{attribute 'linkalways'} 
{attribute 'no_explicit_call' := 'This FB is a CLASS and must be accessed using methods or properties'}
{attribute 'enable_dynamic_creation'}
FUNCTION_BLOCK Dictionary
VAR
	root : I_DictionaryTreeNode;
END_VAR

METHOD PUBLIC AddOrUpdate
VAR_INPUT
	Key : T_MAXSTRING;
	Value : ANY;
END_VAR
root := this^.RecursiveInsert(Key, Value, root);
END_METHOD

METHOD PRIVATE Balance : I_DictionaryTreeNode
VAR_INPUT
	Node : I_DictionaryTreeNode;
END_VAR
VAR
	balanceFactor : DINT;
END_VAR
balanceFactor := THIS^.GetBalanceFactor(Node);

IF (balanceFactor > 1) THEN
  IF (THIS^.getBalanceFactor(Node.left) < 0) THEN
	Node.left := THIS^.leftRotate(Node.left);
  END_IF
  Balance := THIS^.rightRotate(Node);
  RETURN;
END_IF

IF (balanceFactor < -1) THEN
  IF (THIS^.getBalanceFactor(Node.right) > 0) THEN
	Node.right := THIS^.rightRotate(Node.right);
  END_IF
  Balance := THIS^.leftRotate(Node);
  RETURN;
END_IF

Balance := Node;
END_METHOD

METHOD PUBLIC Clear
VAR_INPUT
END_VAR
THIS^.RecursiveClear(root);
root := 0;
END_METHOD

METHOD PUBLIC ContainsKey : BOOL
VAR_INPUT
	Key : T_MAXSTRING;
END_VAR
VAR
	foundNode : I_DictionaryTreeNode;
END_VAR
foundNode := THIS^.RecursiveFind(Key, root);

IF foundNode = 0 THEN
	RETURN;
END_IF

ContainsKey := TRUE;
END_METHOD

METHOD PRIVATE FindMinimum : I_DictionaryTreeNode
VAR_INPUT
	Node : I_DictionaryTreeNode;
END_VAR
VAR
	nextNode : I_DictionaryTreeNode;
END_VAR
nextNode := Node;

WHILE (nextNode.left <> 0) DO
      nextNode := nextNode.left;
END_WHILE;

FindMinimum := nextNode;
END_METHOD

METHOD PRIVATE GetBalanceFactor : DINT
VAR_INPUT
	Node : I_DictionaryTreeNode;
END_VAR
GetBalanceFactor := THIS^.GetHeight(node.left) - THIS^.GetHeight(node.right);
END_METHOD

METHOD PRIVATE GetHeight : DINT
VAR_INPUT
	Node : I_DictionaryTreeNode;
END_VAR
IF Node = 0 THEN
	GetHeight := 0;
	RETURN;
END_IF

GetHeight := Node.Height;
END_METHOD

METHOD PRIVATE LeftRotate : I_DictionaryTreeNode
VAR_INPUT
	Node : I_DictionaryTreeNode;
END_VAR
VAR
	newRoot : I_DictionaryTreeNode;
END_VAR
newRoot := Node.right;
Node.right := newRoot.left;
newRoot.left := Node;
THIS^.UpdateHeight(Node);
THIS^.UpdateHeight(newRoot);
LeftRotate := newRoot;
END_METHOD

METHOD PRIVATE RecursiveClear
VAR_INPUT
	Node : I_DictionaryTreeNode;
END_VAR
IF (Node = 0) THEN
	RETURN;
END_IF

RecursiveClear(Node.Left);
RecursiveClear(Node.Right);
Node.Dispose();
END_METHOD

METHOD PRIVATE RecursiveDelete : I_DictionaryTreeNode
VAR_INPUT
	Key : T_MAXSTRING;
	Node : I_DictionaryTreeNode;
	Parent : I_DictionaryTreeNode;
END_VAR
VAR
	newNode : I_DictionaryTreeNode; 
	parentNode : I_DictionaryTreeNode;
	minValueNode : I_DictionaryTreeNode;
	minValueNodeParent : I_DictionaryTreeNode;
END_VAR
parentNode := Parent;

IF (Node = 0) THEN
	RETURN;
END_IF

IF (Key < Node.Key) THEN
	parentNode := Node;
	Node.left := THIS^.RecursiveDelete(Key, Node.left, parentNode);
ELSIF (Key > Node.Key) THEN
	parentNode := node;
	Node.right := THIS^.RecursiveDelete(Key, Node.right, parentNode);
ELSE 
	// Case 1: Node with only one child or no child
	IF (Node.Left = 0) OR (Node.Right = 0) THEN
		
		IF (Node.Left = 0) THEN
			newNode := Node.Right;
		ELSE
			newNode := Node.Left;
		END_IF
	
		IF (parentNode <> 0) THEN
			IF (parentNode.left = Node) THEN
				parentNode.left := newNode;
			ELSE 
				parentNode.right := newNode;
			END_IF
		END_IF
		
		Node.Dispose();
		RecursiveDelete.Delete := newNode;
		RETURN;
		
	END_IF

	// Case 2: Node with two children
	minValueNode := THIS^.FindMinimum(Node.Right);
	minValueNodeParent := THIS^.RecursiveFindParent(minValueNode.Key, THIS^.root, 0);
	
	IF (minValueNode.Right <> 0) THEN
		minValueNodeParent.Left := minValueNode.Right;
	ELSE 
		minValueNodeParent.Left := 0;
	END_IF
	
	minValueNode.Left := Node.Left;
	minValueNode.Right := Node.Right;
	
	IF (parentNode <> 0) THEN
		IF (parentNode.left = Node) THEN
			parentNode.left := minValueNode;
		ELSE 
			parentNode.right := minValueNode;
		END_IF
	END_IF
	
	Node.Dispose();
	RecursiveDelete.Delete := minValueNode;
	RETURN;
END_IF

THIS^.updateHeight(Node);
RecursiveDelete.Delete := THIS^.balance(Node);
END_METHOD

METHOD PRIVATE RecursiveFind : I_DictionaryTreeNode
VAR_INPUT
	Key : T_MAXSTRING;
	Node : I_DictionaryTreeNode;
END_VAR
IF (Node = 0) THEN
	RETURN;
END_IF

IF (Key < Node.key) THEN
  RecursiveFind := THIS^.RecursiveFind(key, Node.left);
  RETURN;
ELSIF (key > Node.key) THEN
  RecursiveFind := THIS^.RecursiveFind(key, Node.right);
  RETURN;
ELSE 
  RecursiveFind := Node;
  RETURN;
END_IF
END_METHOD

METHOD PRIVATE RecursiveFindParent : I_DictionaryTreeNode
VAR_INPUT
	Key : T_MAXSTRING;
	Node : I_DictionaryTreeNode;
	Parent : I_DictionaryTreeNode;
END_VAR
IF (Node = 0) THEN
	RETURN;
END_IF

IF (Key < Node.Key) THEN
	RecursiveFindParent := THIS^.RecursiveFindParent(Key, Node.Left, Node);
	RETURN;
ELSIF (Key > Node.Key) THEN
	RecursiveFindParent :=  THIS^.RecursiveFindParent(Key, Node.Right, Node);
	RETURN;
ELSE 
	RecursiveFindParent := Parent;
END_IF
END_METHOD

METHOD PRIVATE RecursiveInsert : I_DictionaryTreeNode
VAR_INPUT
	Key : T_MAXSTRING;
	Value : ANY;
	Node : I_DictionaryTreeNode;
END_VAR
VAR
	pAVLTreeNode : POINTER TO DictionaryTreeNode;
END_VAR
IF (Node = 0) THEN
	pAVLTreeNode := __NEW(DictionaryTreeNode);
	pAVLTreeNode^.Initialize(Key, Value);
	RecursiveInsert := pAVLTreeNode^;
	RETURN;
END_IF

IF (Key < node.key) THEN
	Node.left := THIS^.RecursiveInsert(Key, Value, Node.left);
ELSIF (key > node.key) THEN
	Node.right := THIS^.RecursiveInsert(Key, Value, Node.right);
ELSE
	Node.Initialize(Key,Value);
END_IF

THIS^.updateHeight(node);
RecursiveInsert := THIS^.balance(node);
END_METHOD

METHOD PUBLIC Remove
VAR_INPUT
	Key : T_MAXSTRING;
END_VAR
root := THIS^.RecursiveDelete(Key, root, 0);
END_METHOD

METHOD PRIVATE RightRotate : I_DictionaryTreeNode
VAR_INPUT
	Node : I_DictionaryTreeNode;
END_VAR
VAR
	newRoot : I_DictionaryTreeNode;
END_VAR
newRoot := Node.left;
Node.left := newRoot.right;
newRoot.right := Node;
THIS^.UpdateHeight(Node);
THIS^.UpdateHeight(newRoot);
RightRotate := newRoot;
END_METHOD

METHOD PUBLIC TryAdd : BOOL
VAR_INPUT
	Key : T_MAXSTRING;
	Value : ANY;
END_VAR
IF ContainsKey(Key) THEN
	RETURN;
END_IF
	  
THIS^.AddOrUpdate(Key, Value);
TryAdd := TRUE;
END_METHOD

METHOD PUBLIC TryGetValue : BOOL
VAR_INPUT
	Key : T_MAXSTRING;
	Destination	: ANY;
END_VAR
TryGetValue := TryGetValueTo(Key, Destination.pValue, DINT_TO_UDINT(Destination.diSize));
END_METHOD

METHOD PUBLIC TryGetValueTo : BOOL
VAR_INPUT
	Key : T_MAXSTRING;
	DestinationAddress : PVOID;
	DestinationSize : UDINT;
END_VAR
VAR
	foundNode : I_DictionaryTreeNode;
END_VAR
foundNode := THIS^.RecursiveFind(Key, root);

IF foundNode = 0 THEN
	RETURN;
END_IF

TryGetValueTo := foundNode.TryGetTo(DestinationAddress, DestinationSize);
END_METHOD

METHOD PRIVATE UpdateHeight
VAR_INPUT
	Node : I_DictionaryTreeNode;
END_VAR
Node.height := 1 + MAX(THIS^.GetHeight(Node.left), THIS^.GetHeight(Node.right));
END_METHOD

END_FUNCTION_BLOCK

(* stored: Version 1.1.0.1, ProductVersion 3.1.4024.12
   POU Dictionary: Id {031dc881-40c6-4324-9d62-c901951acf8a}, SpecialFunc None
   Folder Private: Id {9d25b7c8-1df3-4ed3-9572-63622da8d884}
   Method AddOrUpdate: Id {570f59cb-7938-4dac-8308-7b97aad37be6}
   Method Balance: Id {de35709f-49a6-4b93-a3ed-80e501fcabee}
   Method Clear: Id {9a75fda3-7d3e-4c00-8099-3ed82d8caa06}
   Method ContainsKey: Id {71cf2ebb-029b-4b77-a924-aa3f84d32e9a}
   Method FindMinimum: Id {4570296d-5467-479c-98b1-7fba065dc91f}
   Method GetBalanceFactor: Id {2a9ce396-eba7-4b31-8293-f5940b4357aa}
   Method GetHeight: Id {7b7a5b98-4d55-42ed-abb9-612f56324af2}
   Method LeftRotate: Id {1e3efb6c-46c1-4085-b7eb-b2d236432957}
   Method RecursiveClear: Id {e76039d0-529f-47ec-a7ab-8c3cbf1105bd}
   Method RecursiveDelete: Id {13a2f8bb-c070-4bfe-a28f-2d1a6438e9b8}
   Method RecursiveFind: Id {72c9c465-18ec-43f4-9bcd-fa5b73279ee3}
   Method RecursiveFindParent: Id {eb8edd98-ca1a-4ae6-8a6d-62c4cf4d7502}
   Method RecursiveInsert: Id {c57d1b55-65c3-4ee8-bbd0-7cf2e85e4be2}
   Method Remove: Id {f7e0145f-426d-4eb3-b5e3-9e9db70ed20a}
   Method RightRotate: Id {8508047b-6b5a-45a7-bfef-30c0ff9ccfee}
   Method TryAdd: Id {0579aed8-c227-47aa-b1a3-1246c4c9910b}
   Method TryGetValue: Id {ffb946e8-f0b7-49b4-a66d-702f84822d81}
   Method TryGetValueTo: Id {aa8e9fd4-2077-48ab-97f4-da34e1392c01}
   Method UpdateHeight: Id {84f1a328-3eec-4abf-9c5a-b520652fa526} *)
